FUNCTION_BLOCK FB_MasterRobot
VAR_INPUT
END_VAR
VAR_OUTPUT
END_VAR
VAR
	// master-slave motion scale
	m_motionScale :LREAL;
	
	// monitor angle
	m_monitorAngle :LREAL;
	
	// master arms, responsible for arm kinematic and control
	m_masterArms :ARRAY[1..g_mArmNum] OF FB_MasterArm;
	
	// arm state
	m_masterArmState:ARRAY[1..g_mArmNum] OF E_masterArmState:=[E_masterArmState.MasterArmState_Init,E_masterArmState.MasterArmState_Init];
	m_lastMasterArmState:ARRAY[1..g_mArmNum] OF E_masterArmState:=[E_masterArmState.MasterArmState_Init,E_masterArmState.MasterArmState_Init];
	m_nextMasterArmState:ARRAY[1..g_mArmNum] OF E_masterArmState:=[E_masterArmState.MasterArmState_Init,E_masterArmState.MasterArmState_Init];
	
	// index(1 to 4) of slave arm which is tele-linked to master arm
	m_teleSlaveArmIdx:ARRAY[1..g_mArmNum] OF E_MatchedSlaveArmIdx:=[MatchedSlaveArmIdx_NULL, MatchedSlaveArmIdx_null];
	
	// all arm controller instance 
	m_armCtrlFactory :ARRAY[1..g_mArmNum,1..MasterArmState_totalNum] OF I_MasterArmCtrl;
	m_armError :ARRAY[1..g_mArmNum] OF FB_ArmError;
	m_armInit :ARRAY[1..g_mArmNum] OF FB_ArmInit;
	m_armHome :ARRAY[1..g_mArmNum] OF FB_ArmHome;
	m_armStandBy :ARRAY[1..g_mArmNum] OF FB_ArmStandBy;
	m_armMatching :ARRAY[1..g_mArmNum] OF FB_ArmMatching;
	m_armReady :ARRAY[1..g_mArmNum] OF FB_ArmReady;
	m_armMasterSlave :ARRAY[1..g_mArmNum] OF FB_ArmMasterSlave;
	m_armClutch :ARRAY[1..g_mArmNum] OF FB_ArmClutch;
	m_armEndoscope :ARRAY[1..g_mArmNum] OF FB_ArmEndoscope;
	m_armCart :ARRAY[1..g_mArmNum] OF FB_ArmCart;
	
	// arm controller interface
	m_armCtrl :ARRAY[1..g_mArmNum] OF I_MasterArmCtrl;
	m_armCtrlCmds :ARRAY[1..g_mArmNum] OF ST_ArmCtrlCmds;

END_VAR

METHOD PUBLIC getStatus : BOOL
VAR_IN_OUT
	// master robot information, including arm status and cartesian data
	r_masterStatus :ST_MasterStatus;
	
	// master robot joint data
	r_masterJointsData :ST_MasterJointData;
	
END_VAR

VAR
	i:INT;
END_VAR
r_masterStatus.m_motionScale := m_motionScale;
r_masterStatus.m_armState:=m_masterArmState;
r_masterStatus.m_teleSlaveArmIdx := m_teleSlaveArmIdx;
FOR i:=1 TO g_mArmNum DO
	// current info
	r_masterStatus.m_gripAngle[i]:=m_masterArms[i].gripAngle;
	// cartesion
	r_masterStatus.m_curArmPose[i]:=m_masterArms[i].curCartPose;
	r_masterStatus.m_curArmTwist[i]:=m_masterArms[i].curCartTwist;
	// joint
	r_masterJointsData.m_curMotorPos[i]:=m_masterArms[i].curMotorPos;
	r_masterJointsData.m_curLinkPos[i]:=m_masterArms[i].curLinkPos;
	r_masterJointsData.m_curJntPos[i]:=m_masterArms[i].curJntPos;
	r_masterJointsData.m_curJntVel[i]:=m_masterArms[i].curJntVel;
	r_masterJointsData.m_curJntTrq[i]:=m_masterArms[i].curJntTrq;
	
	// command info
	// cartesion
	r_masterStatus.m_cmdArmPose[i]:=m_armCtrlCmds[i].m_cmdCartPose;
	r_masterStatus.m_cmdArmTwist[i]:=m_armCtrlCmds[i].m_cmdCartTwist;
	// joint info
	r_masterJointsData.m_cmdJntPos[i]:=m_armCtrlCmds[i].m_cmdJntPos;
	r_masterJointsData.m_cmdJntVel[i]:=m_armCtrlCmds[i].m_cmdJntVel;
	r_masterJointsData.m_cmdJntTrq[i]:=m_armCtrlCmds[i].m_cmdJntTrq;
	
END_FOR
END_METHOD

METHOD PUBLIC Init : BOOL
VAR_INPUT
END_VAR
VAR
	i:INT;
END_VAR
FOR i:=1 TO g_mArmNum DO
	// arm init
	m_masterArms[i].Init(i);
	m_masterArmState[i]:=MasterArmState_Init;
	m_lastMasterArmState[i]:=MasterArmState_Init;
	m_nextMasterArmState[i]:=MasterArmState_Init;
	m_teleSlaveArmIdx[i]:=MatchedSlaveArmIdx_NULL;
	
	// command init
	m_armCtrlCmds[i].m_jntEnableFlag := g_zeroVec7i;
	m_armCtrlCmds[i].m_jntOPMode := g_allPosMode;
	m_armCtrlCmds[i].m_cmdCartPose := m_masterArms[i].curCartPose;
	m_armCtrlCmds[i].m_cmdCartTwist := g_zeroVec6d;
	m_armCtrlCmds[i].m_cmdJntPos := m_masterArms[i].curJntPos;
	m_armCtrlCmds[i].m_cmdJntVel := g_zeroVec7d;
	m_armCtrlCmds[i].m_cmdJntAcc := g_zeroVec7d;
	m_armCtrlCmds[i].m_cmdJntTrq := g_zeroVec7d;
	
	// generate controller factory
	m_armCtrlFactory[i,MasterArmState_Error] := m_armError[i];
	m_armCtrlFactory[i,MasterArmState_Init] := m_armInit[i];
	m_armCtrlFactory[i,MasterArmState_Home] := m_armHome[i];
	m_armCtrlFactory[i,MasterArmState_Standby] := m_armStandBy[i];
	m_armCtrlFactory[i,MasterArmState_Matching] := m_armMatching[i];
	m_armCtrlFactory[i,MasterArmState_Ready] := m_armReady[i];
	m_armCtrlFactory[i,MasterArmState_MasterSlave] := m_armMasterSlave[i];
	m_armCtrlFactory[i,MasterArmState_Clutch] := m_armClutch[i];
	m_armCtrlFactory[i,MasterArmState_Endoscope] := m_armEndoscope[i];
	m_armCtrlFactory[i,MasterArmState_Cart] := m_armCart[i];

	// assign controller
	m_armCtrl[i]:=m_armCtrlFactory[i,m_masterArmState[i]];
END_FOR
END_METHOD

METHOD PUBLIC run : BOOL
VAR_IN_OUT CONSTANT
	i_masterInputDataPool:ST_MasterInputDataPool;
END_VAR
VAR
	i:INT;
END_VAR
m_motionScale := i_masterInputDataPool.m_UIData.m_motionScale;
m_monitorAngle := i_masterInputDataPool.m_cartStatus.m_monitorAngle;

// state machine transition
stateMachine(i_masterInputDataPool);

FOR i:=1 TO g_mArmNum DO
	// update dynamic data
	m_masterArms[i].updateDyna(i_masterInputDataPool.m_masterDynaData.m_massMat[i],
								i_masterInputDataPool.m_masterDynaData.m_gravity[i]);
								
	// update master arm kinematics
	m_masterArms[i].updateStatus();
	
	// null ptr check
	IF 0 = m_armCtrl[i] THEN
		EXIT;
	END_IF
	
	// run controller
	m_armCtrl[i].run(m_monitorAngle, m_teleSlaveArmIdx[i], m_masterArms[i],
						i_masterInputDataPool.m_slaveStatus,m_armCtrlCmds[i]);

	// update commands to drivers
	m_masterArms[i].updateCmds(m_armCtrlCmds[i]);

END_FOR
END_METHOD

// state machine check and transit 
METHOD PROTECTED stateMachine : BOOL
VAR_IN_OUT CONSTANT
		i_masterInputDataPool:ST_MasterInputDataPool;
END_VAR
VAR
	i:INT;
END_VAR
FOR i:=1 TO g_mArmNum DO
	// State machine transit 
	CASE m_masterArmState[i] OF
		// init
		MasterArmState_Init:
			IF m_armCtrl[i].isFinished  THEN
				// NOTICE: multiple cycles joints back to center during initialization
				// 			need to reset joints encoder data again
				m_masterArms[i].initJntPos();
				
				m_nextMasterArmState[i]:=MasterArmState_Home;
			END_IF

		//home
		MasterArmState_Home:
			IF m_armCtrl[i].isFinished  THEN
				m_nextMasterArmState[i]:=MasterArmState_Standby;
			END_IF
		
		//standby
(*		MasterArmState_Standby:
		
		//matching
		MasterArmState_Matching:
		
		//ready
		MasterArmState_Ready:
		
		//MasterSlave
		MasterArmState_MasterSlave:*)
	END_CASE
	
	// Controller transit
	IF m_nextMasterArmState[i]<> m_masterArmState[i] THEN
		// reset current controller
		m_armCtrl[i].reset();
		
		// transit to new one
		m_lastMasterArmState[i]:=m_masterArmState[i];
		m_masterArmState[i]:=m_nextMasterArmState[i];
		m_armCtrl[i]:=m_armCtrlFactory[i,m_masterArmState[i]];
	END_IF
END_FOR
END_METHOD

END_FUNCTION_BLOCK

(* stored: Version 1.1.0.1, ProductVersion 3.1.4024.12
   POU FB_MasterRobot: Id {8cbdb2ba-9735-46e3-8cbc-296330acc8cc}, SpecialFunc None
   Method getStatus: Id {b6139e8c-2703-424c-9761-ad1add6b1ff1}
   Method Init: Id {610a17f3-34c5-4e3c-bbbc-19f9c2f46946}
   Method run: Id {ed6f787a-4dc0-4602-b386-92a3c3880a23}
   Method stateMachine: Id {b9cc8560-9309-49e3-93b5-28cb02b4f5cc} *)
